(* PLC project faults, TNI-Software ControlBuild 4.00.17 *)
(* stored: creationDateTime 2005-06-20T11:54:03-01:00 *)

FUNCTION_BLOCK cmd_equipment_library.faults
  VAR_INPUT  (* CB.group=Orders CB.kind=inputVars *)
    cmd : BOOL := false;  (* CB.libelle=Command of the agitator *)
  END_VAR
  VAR_INPUT  (* CB.group=FeedBacks CB.kind=inputVars *)
    thermalFB : BOOL := false;  (* CB.libelle=Feedback of the thermal protection of the agitator *)
    cmdFB : BOOL := false;  (* CB.libelle=Command feedback *)
  END_VAR
  VAR_INPUT  (* CB.kind=inputVars *)
    acknowledgePB : BOOL := false;  (* CB.libelle=Acknowledgement pushbutton *)
  END_VAR
  VAR_OUTPUT  (* CB.kind=outputVars *)
    generalFault : BOOL := false;  (* CB.mnemonicPatternPropertyName=grlFlt<SY><NU> CB.libelle=General fault of the agitator *)
  END_VAR
  VAR CONSTANT  (* CB.kind=parameterVars *)
    preset : DINT := 2;  (* CB.mnemonicPatternPropertyName=preset<SY><NU> CB.libelle=in seconds *)
  END_VAR
  VAR  (* CB.group=Faults CB.kind=overControlVars *)
    thermalFault : BOOL := false;  (* CB.mnemonicPatternPropertyName=defElec<SY><NU> CB.libelle=Thermal (electric) fault *)
    cmdFBFault : BOOL := false;  (* CB.mnemonicPatternPropertyName=cmdFBFlt<SY><NU> CB.libelle=Command feedback fault *)
  END_VAR

(* LD diagram, written out as Structured Text *)
1:
IF acknowledgePB THEN thermalFault := FALSE; END_IF;
IF acknowledgePB THEN cmdFBFault := FALSE; END_IF;
IF acknowledgePB THEN generalFault := FALSE; END_IF;
2:
ton_sec_1(IN := cmd, PT := preset);
IF ton_sec_1.Q AND NOT cmdFB THEN cmdFBFault := TRUE; END_IF;
3:
ton_sec_2(IN := NOT thermalFB, PT := preset);
IF ton_sec_2.Q THEN thermalFault := TRUE; END_IF;
4:
IF thermalFault OR cmdFBFault THEN generalFault := TRUE; END_IF;
END_FUNCTION_BLOCK
